{attribute 'linkalways'} 
{attribute 'no_explicit_call' := 'This FB is a CLASS and must be accessed using methods or properties'}
{attribute 'enable_dynamic_creation'}
FUNCTION_BLOCK JsonDomNavigator IMPLEMENTS I_JsonPathVisitor
VAR
	jsonDomParser : REFERENCE TO JsonDomParser;
	currentJsonPosition : SJsonValue;
	_currentNode : SJsonValue;
END_VAR

METHOD ArrayIndexFound
VAR_INPUT
	Index : UDINT;
END_VAR
currentJsonPosition := jsonDomParser.GetArrayValueByIdx(currentJsonPosition, Index);
END_METHOD

PROPERTY PUBLIC CurrentNode : SJsonValue
GET
CurrentNode := _currentNode;
END_GET
END_PROPERTY

METHOD EndOfParse
VAR_INPUT
END_VAR
_currentNode := currentJsonPosition;
END_METHOD

METHOD FB_init : BOOL
VAR_INPUT
	bInitRetains : BOOL; // if TRUE, the retain variables are initialized (warm start / cold start)
	bInCopyCode : BOOL;  // if TRUE, the instance afterwards gets moved into the copy code (online change)
	JsonDomParser : REFERENCE TO JsonDomParser;
END_VAR
THIS^.jsonDomParser REF= JsonDomParser;
END_METHOD

METHOD InvalidSyntaxFound
VAR_INPUT
	Character : BYTE;
	Position : UDINT;
END_VAR
currentJsonPosition := 0;
END_METHOD

METHOD PropertyFound
VAR_INPUT
	Name : T_MAXSTRING;
END_VAR
currentJsonPosition := jsonDomParser.FindMember(currentJsonPosition,Name);
END_METHOD

METHOD StartOfParse
VAR_INPUT
END_VAR
currentJsonPosition := jsonDomParser.GetDocumentRoot();
END_METHOD

END_FUNCTION_BLOCK

(* stored: Version 1.1.0.1, ProductVersion 3.1.4024.12
   POU JsonDomNavigator: Id {8dcae62e-8322-46a6-945f-bd6da2ebb110}, SpecialFunc None
   Folder Constructor: Id {04fc1430-9345-473f-a4b2-f1c612665b3e}
   Method ArrayIndexFound: Id {98db7489-e8e0-4d0a-a655-8d7a75b6cd7b}
   Property CurrentNode: Id {989a9abf-47c4-46fe-8239-df8a3794c12b}
   Get Get: Id {10905a16-4fee-402f-a2c3-6b5973ef1cdb}
   Method EndOfParse: Id {1933187d-055b-4280-a3dd-fb95e40be1c4}
   Method FB_init: Id {c9de5196-45a9-4bb9-8cd3-1c3a220960f4}
   Method InvalidSyntaxFound: Id {00a8c3f8-bf0b-456e-8b7d-b3d7e64b3294}
   Method PropertyFound: Id {0373e239-39fc-45b6-a1bd-230ceca8166d}
   Method StartOfParse: Id {2a485667-84fd-4586-9186-faf843b7ab5e} *)
